// TIA Portal project "3M - N (2)" (V16)

(* hardware
DEVICE "S7-1200 station_1"  S7-1200 Station
   slot 0: "Rack_0"  S7-1200 Rack  Rack  V1.0
   slot 1: "PLC_1"  CPU 1212C AC/DC/Rly  6ES7 212-1BE40-0XB0  V4.0
*)

// ===== PLC "PLC_1"  CPU 1212C AC/DC/Rly =====

VAR_GLOBAL   // PLC tag table "Default tag table"
   "start1" AT %I0.2 : Bool;
   "K1" AT %Q0.0 : Bool;
   "stop1" AT %I0.4 : Bool;
   "k2" AT %Q0.1 : Bool;
   "STOP" AT %I0.3 : Bool;
   "T1 tag" AT %M0.0 : Bool;
   "T2 tag" AT %M0.1 : Bool;
   "X" AT %M0.2 : Bool;
   "C1" AT %M1.0 : Bool;
   "C2" AT %M1.1 : Bool;
   "K3" AT %Q0.2 : Bool;
   "C3" AT %M1.2 : Bool;
   "C4" AT %M1.3 : Bool;
   "T3 tag" AT %M0.3 : Bool;
   "Tag_1" AT %M0.6 : Bool;
   "Tag_2" AT %M2.0 : Bool;
   "2nd cycle" AT %M2.1 : Bool;
   "Tag_3" AT %M2.3 : Bool;
   "Tag_4" AT %M3.2 : Bool;
END_VAR

// folder: System blocks/Program resources

DATA_BLOCK "T1"   // DB2
{ S7_Optimized_Access := 'TRUE' }
AUTHOR : Simatic
FAMILY : IEC
NAME : IEC_TMR
VERSION : 1.0
// stored: InstanceOfName IEC_TIMER
"IEC_TIMER"
BEGIN
END_DATA_BLOCK

DATA_BLOCK "TON1"   // DB3
{ S7_Optimized_Access := 'TRUE' }
AUTHOR : Simatic
FAMILY : IEC
NAME : IEC_TMR
VERSION : 1.0
// stored: InstanceOfName IEC_TIMER
"IEC_TIMER"
BEGIN
END_DATA_BLOCK

DATA_BLOCK "T3"   // DB4
{ S7_Optimized_Access := 'TRUE' }
AUTHOR : Simatic
FAMILY : IEC
NAME : IEC_TMR
VERSION : 1.0
// stored: InstanceOfName IEC_TIMER
"IEC_TIMER"
BEGIN
END_DATA_BLOCK

// folder: (top level)

ORGANIZATION_BLOCK "Main"   // OB1, LAD, ProgramCycle
TITLE = "Main Program Sweep (Cycle)"
{ S7_Optimized_Access := 'TRUE' }
VERSION : 0.1
   VAR_INPUT
      Initial_Call : Bool;   // Initial call of this OB
      Remanence : Bool;   // =True, if remanent data are available
   END_VAR
   VAR_TEMP   // added for the SCL form of the ladder/FBD networks
      _w1 : Bool;
   END_VAR
BEGIN

REGION Network 1: start
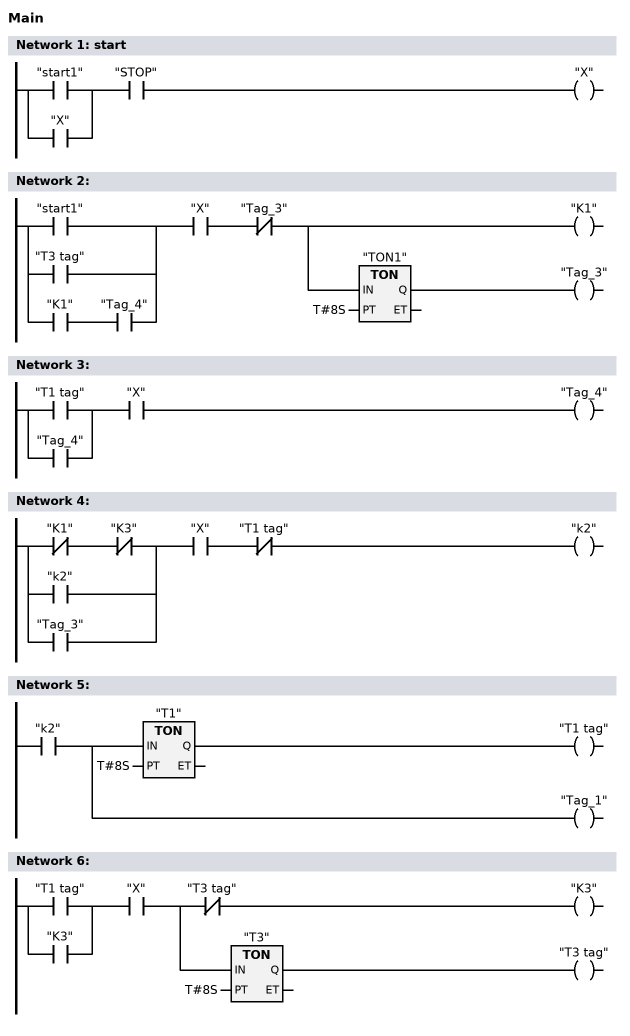
   RUNG wire#powerrail
      Contact( "start1" )
      wire#w1
      Contact( "STOP" )
      Coil( "X" )
   END_RUNG
   RUNG wire#powerrail
      Contact( "X" )
   END_RUNG wire#w1
   // the same network as SCL:
   "X" := ("start1" OR "X") AND "STOP";
END_REGION

REGION Network 2
   "K1" := ("start1" OR "T3 tag" OR ("K1" AND "Tag_4")) AND "X" AND NOT "Tag_3";
   "TON1".TON(IN := "K1", PT := T#8S);
   "Tag_3" := "TON1".Q;
END_REGION

REGION Network 3
   RUNG wire#powerrail
      Contact( "T1 tag" )
      wire#w1
      Contact( "X" )
      Coil( "Tag_4" )
   END_RUNG
   RUNG wire#powerrail
      Contact( "Tag_4" )
   END_RUNG wire#w1
   // the same network as SCL:
   "Tag_4" := ("T1 tag" OR "Tag_4") AND "X";
END_REGION

REGION Network 4
   RUNG wire#powerrail
      I_Contact( "K1" )
      I_Contact( "K3" )
      wire#w1
      Contact( "X" )
      I_Contact( "T1 tag" )
      Coil( "k2" )
   END_RUNG
   RUNG wire#powerrail
      Contact( "k2" )
   END_RUNG wire#w1
   RUNG wire#powerrail
      Contact( "Tag_3" )
   END_RUNG wire#w1
   // the same network as SCL:
   "k2" := ((NOT "K1" AND NOT "K3") OR "k2" OR "Tag_3") AND "X" AND NOT "T1 tag";
END_REGION

REGION Network 5
   "T1".TON(IN := "k2", PT := T#8S);
   "T1 tag" := "T1".Q;
   "Tag_1" := "k2";
END_REGION

REGION Network 6
   #_w1 := ("T1 tag" OR "K3") AND "X";
   "K3" := #_w1 AND NOT "T3 tag";
   "T3".TON(IN := #_w1, PT := T#8S);
   "T3 tag" := "T3".Q;
END_REGION
END_ORGANIZATION_BLOCK